FUNCTION_BLOCK LinearContinuousDrive_2Sensor EXTENDS FBA_LinearDrive IMPLEMENTS I_LinearContinuousDrive
VAR_INPUT
	drive : I_ContinuousDrive;
END_VAR
VAR
	extendLimit AT %I* : BOOL;
END_VAR

override();

ready := bEnable AND NOT Active AND HomeSet;

PROPERTY Active : BOOL
GET
Active := drive.Active;
END_GET
END_PROPERTY

PROPERTY AtExtendLimit : BOOL
GET
AtExtendLimit := extendLimit <> sensorDefaultState;
END_GET
END_PROPERTY

PROPERTY Error : BOOL
GET
error := drive.Error;
END_GET
END_PROPERTY

METHOD homingSequence : BOOL
(*
homing sequence is different for linear motion devices with limit sensors
*)
CASE step OF
	Homing.IDLE:
		reset();
		IF bEnable THEN
			step := Homing.START;
		END_IF
		
	Homing.START:
		IF AtHome THEN
			step := Homing.STOP;
			
		ELSIF AtExtendLimit THEN
			step := Homing.RETRY;
			
		ELSE
			moveContinuous(newDirection:= MC_Positive_Direction);
		END_IF
		
	Homing.STOP:
		IF stop() THEN
			step := Homing.DONE;
		END_IF
		
	Homing.DONE:
		homingComplete := TRUE;
		step := Homing.IDLE;
		
END_CASE
END_METHOD

METHOD moveContinuous : BOOL
VAR_INPUT
	newDirection : MC_Direction;
END_VAR
drive.moveContinuous(newDirection:= newDirection);

direction := newDirection;
END_METHOD

METHOD PRIVATE override : BOOL
VAR_INPUT
END_VAR
(*
-at home and attempting to traverse outward
-at outer limit and attempting to traverse outward
-at inner limit and attempting to traverse inwards
*)
(*
inward = negative direction, negative velocity
outward = positive direction, positive velocity
*)

IF error THEN
	stop();
	reset();
	
ELSIF
	(AtExtendLimit AND direction = MC_Negative_Direction) OR
	(AtHome AND direction = MC_Positive_Direction)
THEN
	stop();
END_IF
END_METHOD

METHOD reset : BOOL
VAR_INPUT
END_VAR
reset := drive.reset();
END_METHOD

METHOD stop : BOOL
VAR_INPUT
END_VAR
stop := drive.stop();
END_METHOD

METHOD toHome : BOOL
VAR_INPUT
END_VAR
IF AtHome THEN
	toHome := TRUE;
ELSE
	moveContinuous(newDirection := MC_Negative_Direction);
END_IF
END_METHOD

END_FUNCTION_BLOCK

(* stored: Version 1.1.0.1, ProductVersion 3.1.4024.11
   POU LinearContinuousDrive_2Sensor: Id {2d9188cd-ad30-4956-8d5f-b88d3102c3fe}, SpecialFunc None
   Folder Private: Id {3ba3509b-0d40-4ea4-811a-947a630516e4}
   Folder Properties: Id {7dd186fb-ba85-4c59-a970-19a54fcfadc2}
   Property Active: Id {088c139b-6a0c-4f65-8518-00f9c8339a6d}
   Get Get: Id {335bcb3e-d6ec-4644-aa30-191dfa882793}
   Property AtExtendLimit: Id {8f1e0ffe-cd76-400b-89c9-ab58ba076ac4}
   Get Get: Id {152a49a6-c78f-4963-b6d1-a7f0a31eada4}
   Property Error: Id {5b1c6a70-d5d5-4300-b867-3ef3d15fb7ac}
   Get Get: Id {ee9054dc-d07d-462c-a839-fe09eb0253e9}
   Method homingSequence: Id {bfcd0096-7833-4bef-97f6-250bc428dc2f}
   Method moveContinuous: Id {af100d6f-af7e-4519-9823-440dfe81e2d5}
   Method override: Id {0e3ca204-a9dd-467c-8642-994a01b39513}
   Method reset: Id {d507b5af-49fc-4f61-bfe7-b2cbe9255b70}
   Method stop: Id {cd4bebce-eaf2-4b90-8156-811ca27572dd}
   Method toHome: Id {1bee4eb9-8f8f-4283-b2d6-695b63df7300} *)
